PROGRAM MAIN
VAR
	LocalEtherCATDevState	AT%I*:UINT ;
END_VAR

PRG_EncoderSim();

PRG_AnalogSim();

END_PROGRAM

(* stored: Version 1.1.0.1, ProductVersion 3.1.4024.11
   POU MAIN: Id {c90d7607-1feb-46bb-9bc2-7b1fb026a69c}, SpecialFunc None *)
